FUNCTION_BLOCK intValueChange (* Basic Function Block Type *)
  (* Standard: 61499-2 *)
  (* Version 0.0, 31/08/2026, Template *)
  PACKAGE Hidryco.HidrycoLib;
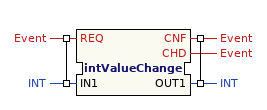
  EVENT_INPUT
    REQ WITH IN1; (* Normal Execution Request *)
  END_EVENT
  EVENT_OUTPUT
    CNF WITH OUT1; (* Execution Confirmation *)
    CHD;
  END_EVENT
  VAR_INPUT
    IN1 : INT; (* Argument *)
  END_VAR
  VAR_OUTPUT
    OUT1 : INT; (* Result *)
  END_VAR
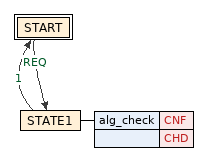
  EC_STATES
    START; (* Initial State *)
    STATE1 : alg_check -> CNF, -> CHD;
  END_STATES
  EC_TRANSITIONS
    START TO STATE1 := REQ;
    STATE1 TO START := 1;
  END_TRANSITIONS
  ALGORITHM alg_check IN ST:
CHD := OUT1 <> IN1;

OUT1 := IN1;

;
  END_ALGORITHM
END_FUNCTION_BLOCK
